///EL2088 | 8-channel digital output terminal 24 V DC, 0.5 A, negative switching
FUNCTION_BLOCK EL2088

VAR_INPUT
	En: BOOL;
	bDo_1: BOOL;
	bDo_2: BOOL;
	bDo_3: BOOL;
	bDo_4: BOOL;
	bDo_5: BOOL;
	bDo_6: BOOL;
	bDo_7: BOOL;
	bDo_8: BOOL;
	iTerminal_ID : INT;
	ErrorSystem : POINTER TO ST_ErrorSystem;
END_VAR

VAR_OUTPUT
	EnO: BOOL;
	bError: BOOL;
END_VAR

VAR
	Channel_1_Output AT %Q*: BOOL;
	Channel_2_Output AT %Q*: BOOL;
	Channel_3_Output AT %Q*: BOOL;
	Channel_4_Output AT %Q*: BOOL;
	Channel_5_Output AT %Q*: BOOL;
	Channel_6_Output AT %Q*: BOOL;
	Channel_7_Output AT %Q*: BOOL;
	Channel_8_Output AT %Q*: BOOL;
	WcState_WcState AT %I*: BOOL;
	InfoData_State AT %I*: UINT;
	
	//FB-s
	EL2088_Error : FB_TerminalError;
END_VAR

EnO:=En;

//Error FB instance
EL2088_Error(
	En := TRUE,
	iTerminal_ID := iTerminal_ID,
	bWcState := WcState_WcState,
	uiInfoData_State := InfoData_State,
	pErrorSystem := ErrorSystem,
	bError => bError,
);

IF En THEN
	IF bError=FALSE THEN
		Channel_1_Output:=bDo_1;
		Channel_2_Output:=bDo_2;
		Channel_3_Output:=bDo_3;
		Channel_4_Output:=bDo_4;
		Channel_5_Output:=bDo_5;
		Channel_6_Output:=bDo_6;
		Channel_7_Output:=bDo_7;
		Channel_8_Output:=bDo_8;
	END_IF
END_IF

END_FUNCTION_BLOCK

(* stored: Version 1.1.0.1, ProductVersion 3.1.4022.10
   POU EL2088: Id {e8393d2e-b70b-42b8-a453-a029acf3fc5b}, SpecialFunc None *)
